{region '#Template'}
	{attribute 'Version' := '5.0.0.0'}
	{attribute 'Tags' := '"LCID": "1031", "Text": "RA, Beleuchtung, Anwenderfunktionen, Konstantlicht"'}
	{attribute 'Tags' := '"LCID": "1033", "Text": "RA, Lighting, User-functions, constant light control"'}
	{attribute 'Using' := '"Type": "Template", "URI": "ST_BA_LightActuatorFeedback"'}
	{attribute 'Description' := '"LCID": "1031", "Text": "Beleuchtung Konstantlichtregelung"'}
	{attribute 'Description' := '"LCID": "1033", "Text": "Lighting constant light control"'}
{endregion}
FUNCTION_BLOCK FB_BA_LightGroupConstant EXTENDS FB_BA_Ext_LightConstCtrl
VAR_INPUT
	bManualSwitch			: BOOL;
	bOn						: BOOL;
	bOff					: BOOL;
	bResetRoomFunction		: BOOL;			// inactivates the whole function: control-mode AND manual-mode
	bPresence				: BOOL;
	fBrightness				: REAL;
	                        
	stAreaLighting			: ST_BA_Lighting;
	stScene					: ST_BA_Lighting;
	stReferenceFeedback		: ST_BA_LightActuatorFeedback;
	                        
END_VAR                     
                            
VAR_OUTPUT                  
	stLighting				: ST_BA_Lighting;
	bAdjusting				: BOOL;				// This signal is to be used to poll the brightness faster in case of a fieldbus-based brightness-sensor
END_VAR

		
VAR_INPUT CONSTANT PERSISTENT				
	fHys 					: REAL;				// constant light: hysteresis for control-deviation. Limited from 0 to rBrtns
	{attribute 'parameterUnit':= 'ms'}          
	nSwiOvrTi				: UDINT;			// distinction time [ms] between short click and long-press
	{attribute 'parameterUnit':= 's'}       	
	nSwiTi					: UDINT;			// switch-ramp-time [s] to drive rOut from 0 to 100 
	{attribute 'parameterUnit':= 's'}       	
	nDimTi					: UDINT;			// dim-ramp-time [s] to drive rOut from 0 to 100 
	{attribute 'parameterUnit':= 's'}       	
	nRampTi					: UDINT;			// constant light: control-ramp-time [s]
	{attribute 'parameterUnit':= 's'}           
	nPreOffRampTi			: UDINT;			// ramp time [s] for the pre-off-function
	{attribute 'parameterUnit':= 's'}       	
	nBrtnsAdjTi				: UDINT;			// constant light: time [s] to let the brighness sensor adjust to new values before taking them over to the internal control
	{attribute 'parameterUnit':= '%'}           
	fOnValCtrl				: REAL;				// on value in control mode, limited from 0 to 100.
	{attribute 'parameterUnit':= '%'}           
	fOnValMan				: REAL;				// on value in memory mode, limited from 0 to 100.
	{attribute 'parameterUnit':= '%'}           
	fPreOffVal				: REAL;				// light value on pre-off-delay period.
	{attribute 'parameterUnit':= 's'}           
	nPreOffDly				: UDINT;			// duration [s] of pre-off-delay period
	{attribute 'parameterUnit':= '%'}           
	fMinVal 				: REAL;				// constant light: minimum control-value before the light control wants to turn off
	{attribute 'parameterUnit':= 's'}           
	nMinOffDly 				: UDINT;			// constant light: time [s] before switching off at fMinVal
	{attribute 'parameterUnit':= 's'}           
	nMinOnDly 				: UDINT;			// constant light: time [s] before switching on at fMinVal
	bMemoryMode				: BOOL;				// memory mode. switch on to value before last off	
	{attribute 'parameterUnit':= 'KELVIN'}	                    
	fLgtT					: REAL		:= 3000;	
END_VAR	
		             
VAR_INPUT CONSTANT           	
	SpBrightness			: FB_BA_AV_Op;
	ManMode					: FB_BA_LightingEvt :=( ePrio:= E_BA_LightingPrio.eManual);	
	CnstLgtAuto				: FB_BA_LightingEvt :=( ePrio:= E_BA_LightingPrio.eAutomaticLight);
END_VAR
VAR
	ConstLgtCtrl			: FB_BA_LightCtrlConst;	
	PrioSwi					: FB_BA_LightingTgmSel4;	
END_VAR

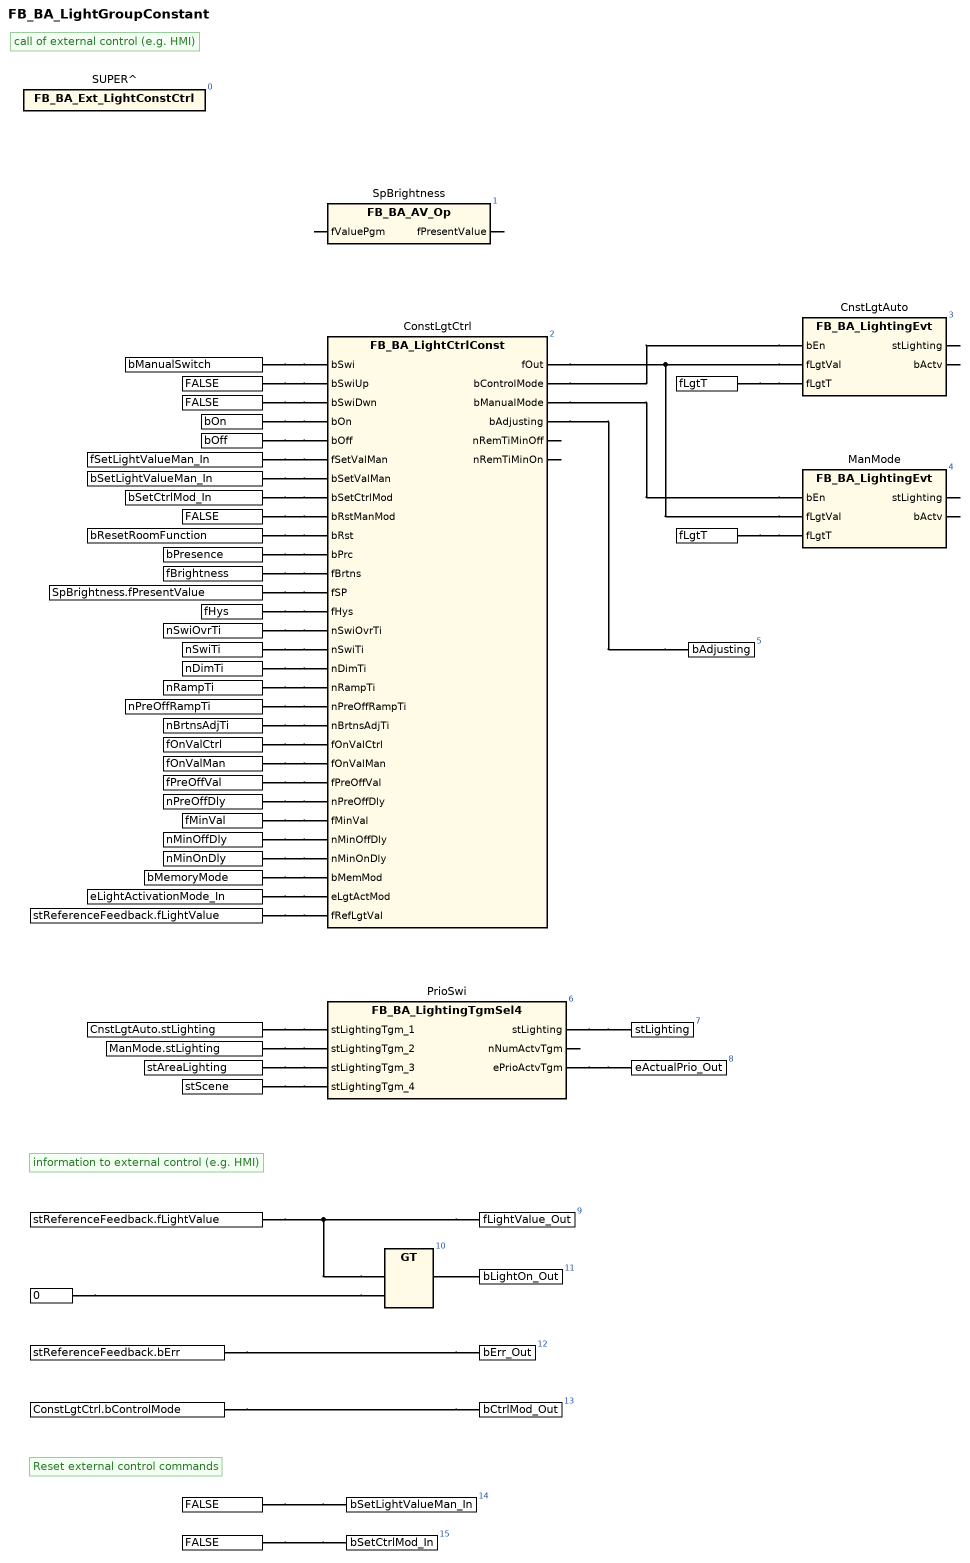
// call of external control (e.g. HMI)
SUPER^(); // FB_BA_Ext_LightConstCtrl
SpBrightness(); // FB_BA_AV_Op
ConstLgtCtrl(
    bSwi := bManualSwitch,
    bSwiUp := FALSE,
    bSwiDwn := FALSE,
    bOn := bOn,
    bOff := bOff,
    fSetValMan := fSetLightValueMan_In,
    bSetValMan := bSetLightValueMan_In,
    bSetCtrlMod := bSetCtrlMod_In,
    bRstManMod := FALSE,
    bRst := bResetRoomFunction,
    bPrc := bPresence,
    fBrtns := fBrightness,
    fSP := SpBrightness.fPresentValue,
    fHys := fHys,
    nSwiOvrTi := nSwiOvrTi,
    nSwiTi := nSwiTi,
    nDimTi := nDimTi,
    nRampTi := nRampTi,
    nPreOffRampTi := nPreOffRampTi,
    nBrtnsAdjTi := nBrtnsAdjTi,
    fOnValCtrl := fOnValCtrl,
    fOnValMan := fOnValMan,
    fPreOffVal := fPreOffVal,
    nPreOffDly := nPreOffDly,
    fMinVal := fMinVal,
    nMinOffDly := nMinOffDly,
    nMinOnDly := nMinOnDly,
    bMemMod := bMemoryMode,
    eLgtActMod := eLightActivationMode_In,
    fRefLgtVal := stReferenceFeedback.fLightValue); // FB_BA_LightCtrlConst
CnstLgtAuto(bEn := ConstLgtCtrl.bControlMode, fLgtVal := ConstLgtCtrl.fOut, fLgtT := fLgtT); // FB_BA_LightingEvt
ManMode(bEn := ConstLgtCtrl.bManualMode, fLgtVal := ConstLgtCtrl.fOut, fLgtT := fLgtT); // FB_BA_LightingEvt
bAdjusting := ConstLgtCtrl.bAdjusting;
PrioSwi(
    stLightingTgm_1 := CnstLgtAuto.stLighting,
    stLightingTgm_2 := ManMode.stLighting,
    stLightingTgm_3 := stAreaLighting,
    stLightingTgm_4 := stScene); // FB_BA_LightingTgmSel4
stLighting := PrioSwi.stLighting;
eActualPrio_Out := PrioSwi.ePrioActvTgm;
fLightValue_Out := stReferenceFeedback.fLightValue;
// information to external control (e.g. HMI)
bLightOn_Out := stReferenceFeedback.fLightValue > 0;
bErr_Out := stReferenceFeedback.bErr;
bCtrlMod_Out := ConstLgtCtrl.bControlMode;
// Reset external control commands
bSetLightValueMan_In := FALSE;
bSetCtrlMod_In := FALSE;

METHOD FB_init : BOOL
VAR_INPUT
	bInitRetains : BOOL; // if TRUE, the retain variables are initialized (warm start / cold start)
	bInCopyCode : BOOL;  // if TRUE, the instance afterwards gets moved into the copy code (online change)
END_VAR
SpBrightness.iParent		:= THIS^;
SpBrightness.iLabel			:= LblFun_Setpoint;
SpBrightness.eUnit			:= E_BA_Unit.eLight_Luxes;  
SpBrightness.fValueRm		:= 300.0;
SpBrightness.fCOVIncrement	:= BA2_Param.fDefCOVIncrement;	

fHys 						:= 50;		// constant-light: hysteresis for control-deviation [lux].
nSwiOvrTi					:= 250;		// distinction-time [ms] between short-lick and long-press
nSwiTi						:= 2;		// switch-ramp-time [s] to drive rOut from 0 to 100 
nDimTi						:= 10;		// dim-ramp-time [s] to drive rOut from 0 to 100 
nRampTi						:= 60;		// constant-light: control-ramp-time [s]
nPreOffRampTi				:= 2;		// ramp-time [s] for the pre-off-function
nBrtnsAdjTi					:= 5;		// constant-light: time [s] to let the brighness-sensor adjust to new values before taking them over to the internal control
fOnValCtrl					:= 50;		// on-Value, limited from 0 to 100.
fOnValMan					:= 100;		// on-Value, limited from 0 to 100.
fPreOffVal					:= 4;		// light-value on pre-off-delay period.
nPreOffDly					:= 10;		// duration [s] of pre-off-delay period
fMinVal 					:= 4;		// constant-light: minimum control-value before the light control wants to turn off
nMinOffDly 					:= 300;		// constant-light: time [s] before switching off at fMinVal
nMinOnDly 					:= 300;		// constant-light: time [s] before switching on at fMinVal
bMemoryMode					:= FALSE;	// memory-mode. switch on to value before last off

fLgtT						:= 3000;			// [K]
END_METHOD

END_FUNCTION_BLOCK

(* stored: Version 1.1.0.1, ProductVersion 3.1.4024.12
   POU FB_BA_LightGroupConstant: Id {17277180-4e36-4c68-90df-1ec53ed3aecc}, SpecialFunc None
   Method FB_init: Id {a13273b9-3214-497f-b561-684a682bb998} *)
